PROGRAM Measurement_Angle_Offset
VAR
END_VAR

astAxes[AXIS_MEASUREMENT_ANGLE_OFFSET].stInputs.bLimitBwd := TRUE;
astAxes[AXIS_MEASUREMENT_ANGLE_OFFSET].stInputs.bLimitFwd := TRUE;
astAxes[AXIS_MEASUREMENT_ANGLE_OFFSET].stControl.bEnable:= TRUE;

END_PROGRAM

(* stored: Version 1.1.0.1, ProductVersion 3.1.4024.11
   POU Measurement_Angle_Offset: Id {87603760-826b-4313-a4cd-b2f0401911a5}, SpecialFunc None *)
